// TIA Portal project "Bachelor GIT Project" (V17)

(* hardware
DEVICE "S7-1500/ET200MP station_1"  S7-1500 station
   slot 0: "Rail_0"  Rack  6ES7 590-1***0-0AA0
   slot 1: "PLC_1"  CPU 1511-1 PN  6ES7 511-1AK00-0AB0  V1.8
      slot 3: "CPU display_1"  6ES7591-1AA00-0AA0
      slot 32768: "PROFINET interface_1"  X1
         slot 32769: "Port_1"  X1 P1
         slot 32770: "Port_2"  X1 P2
DEVICE "HMI_1"  TP1200 Comfort PRO
   slot 0: "HMI_1"  TP1200 Comfort PRO  6AV2 124-0MC24-0AXx  17.0.0.0
   slot 1: "HMI_RT_1"  TP1200 Comfort PRO  6AV2 124-0MC24-0AXx  17.0.0.0
   slot 5: "HMI_1.IE_CP_1"  PROFINET Interface  17.0.0.0
      slot 1: "PROFINET Interface_1"  PROFINET Interface
         slot 1: "Port_1"  Port
         slot 2: "Port_2"  Port
   slot 6: "HMI_1.IE_CP_2"  PROFINET Interface  17.0.0.0
      slot 1: "PROFINET Interface_GBit"  PROFINET Interface
         slot 1: "Port_1"  Port
   slot 7: "HMI_1.MPI/DP_CP_1"  MPI/DP Interface  17.0.0.0
*)

// ===== PLC "PLC_1"  CPU 1511-1 PN =====

VAR_GLOBAL   // PLC tag table "Digital"
   "DigitalInput" AT %I0.0 : Bool;
   "DigitalOutput" AT %I0.1 : Bool;
END_VAR

VAR_GLOBAL   // PLC tag table "Analog"
   "AnalogInput" AT %QW0 : Int;
   "AnalogOutput" AT %IW0 : Int;
END_VAR

DATA_BLOCK "DataBlock"   // DB1
{ S7_Optimized_Access := 'TRUE' }
VERSION : 0.1
   VAR
      Speed_DB : Int;
      Input : Int;
      Output : Real;
   END_VAR
BEGIN
END_DATA_BLOCK

FUNCTION "Speed_SCL" : Void   // FC1, SCL
{ S7_Optimized_Access := 'TRUE' }
VERSION : 0.1
   VAR_TEMP
      Speed : Bool;
      Speed_Var2 : Bool;
   END_VAR
BEGIN

   IF #Speed_Var2 AND #Speed = TRUE THEN
       #Speed := TRUE;
       #Speed := TRUE;
   END_IF;
END_FUNCTION

FUNCTION "Speed_LAD" : Void   // FC2, LAD
{ S7_Optimized_Access := 'TRUE' }
VERSION : 0.1
   VAR_TEMP
      Speed : Bool;
      Speed_Var : Bool;
   END_VAR
BEGIN

REGION Network 1
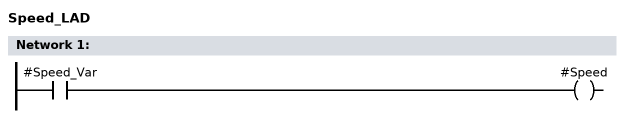
   RUNG wire#powerrail
      Contact( #Speed_Var )
      Coil( #Speed )
   END_RUNG
   // the same network as SCL:
   #Speed := #Speed_Var;
END_REGION
END_FUNCTION

FUNCTION "ScalingAnalogInput" : Void   // FC3, LAD
{ S7_Optimized_Access := 'TRUE' }
   VAR_INPUT
      RawValue : Int;
   END_VAR
   VAR_OUTPUT
      Output : Real;
   END_VAR
   VAR_TEMP
      Value : Real;
   END_VAR
BEGIN

REGION Network 1
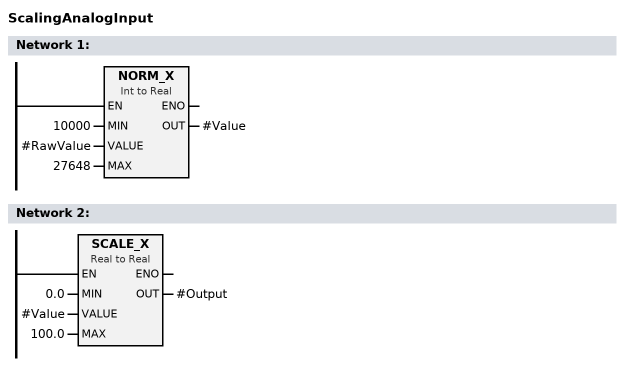
   RUNG wire#powerrail
      { S7_Templates := "[SrcType := Int, DestType := Real]" } Normalize(min := 10000, value := #RawValue, max := 27648, out => #Value)
   END_RUNG
   // the same network as SCL:
   #Value := NORM_X(MIN := 10000, VALUE := #RawValue, MAX := 27648);
END_REGION

REGION Network 2
   RUNG wire#powerrail
      { S7_Templates := "[SrcType := Real, DestType := Real]" } Scale(min := 0.0, value := #Value, max := 100.0, out => #Output)
   END_RUNG
   // the same network as SCL:
   #Output := SCALE_X(MIN := 0.0, VALUE := #Value, MAX := 100.0);
END_REGION
END_FUNCTION

ORGANIZATION_BLOCK "Main"   // OB1, LAD, ProgramCycle
TITLE = "Main Program Sweep (Cycle)"
{ S7_Optimized_Access := 'TRUE' }
VERSION : 0.1
   VAR_INPUT
      Initial_Call : Bool;   // Initial call of this OB
      Remanence : Bool;   // =True, if remanent data are available
   END_VAR
BEGIN

REGION Network 1
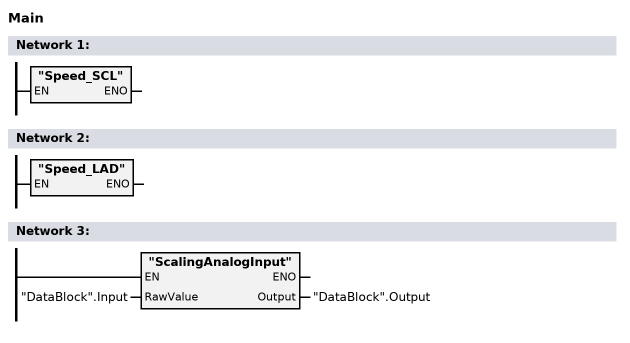
   RUNG wire#powerrail
      "Speed_SCL"()
   END_RUNG
   // the same network as SCL:
   "Speed_SCL"();
END_REGION

REGION Network 2
   RUNG wire#powerrail
      "Speed_LAD"()
   END_RUNG
   // the same network as SCL:
   "Speed_LAD"();
END_REGION

REGION Network 3
   RUNG wire#powerrail
      "ScalingAnalogInput"(RawValue := "DataBlock".Input, Output => "DataBlock".Output)
   END_RUNG
   // the same network as SCL:
   "ScalingAnalogInput"(RawValue := "DataBlock".Input, Output => "DataBlock".Output);
END_REGION
END_ORGANIZATION_BLOCK

(* ===== HMI "HMI_RT_1" =====
system functions are stored by id; their names below are inferred from use
connection "HMI_Connection_1": ETHERNET, S7_1500_OMS

HMI tags "Default tag table"
   "Tag_ScreenNumber" : UInt, internal

screen "Root screen" 1280x740, template "Template_1"
   on GenerateScreen: SetTag("Tag_ScreenNumber", 1)
   TextField "HmiScreenItemData" at 128,324 size 1024x27; Text 'Welcome to HMI_1 (TP1200 Comfort PRO)!'

Template "Template_1" 1280x740
   Button "Exit" at 1200,679 size 78x59; TextOff 'Exit'; PictureOff "ExitRuntime_TP1200_Comfort_PRO_TR"; PictureOn "ExitRuntime_TP1200_Comfort_PRO_TR"
      on Release: StopRuntime(0)
   Button "Template_Button" at 1120,679 size 78x59; TextOff 'Text'
   Button "Template_Button_1" at 1040,679 size 78x59; TextOff 'Text'
   Button "Template_Button_2" at 960,679 size 78x59; TextOff 'Text'
   Button "Template_Button_3" at 880,679 size 78x59; TextOff 'Text'
   Button "Template_Button_4" at 800,679 size 78x59; TextOff 'Text'
   Button "Template_Button_5" at 720,679 size 78x59; TextOff 'Text'
   Button "Template_Button_6" at 640,679 size 78x59; TextOff 'Text'
   Button "Template_Button_7" at 561,679 size 78x59; TextOff 'Text'
   Button "Template_Button_8" at 481,679 size 78x59; TextOff 'Text'
   Button "Template_Button_9" at 401,679 size 78x59; TextOff 'Text'
   Button "Template_Button_10" at 321,679 size 78x59; TextOff 'Text'
   Button "Template_Button_11" at 241,679 size 78x59; TextOff 'Text'
   Button "Template_Button_12" at 161,679 size 78x59; TextOff 'Text'
   Button "Alarms" at 81,679 size 78x59; TextOff 'Alarms'; PictureOff "AlarmDisplay_TP1200_Comfort_PRO_TR"; PictureOn "AlarmDisplay_TP1200_Comfort_PRO_TR"
      on Release: function_ef3f5d25("Alarm window_Unacknowledged", -1)
   Button "Start screen" at 1,679 size 78x59; TextOff 'Start screen'; PictureOff "NavigateHome_TP1200_Comfort_PRO_TR"; PictureOn "NavigateHome_TP1200_Comfort_PRO_TR"
      on Release: ActivateScreen("Root screen", 0)
*)